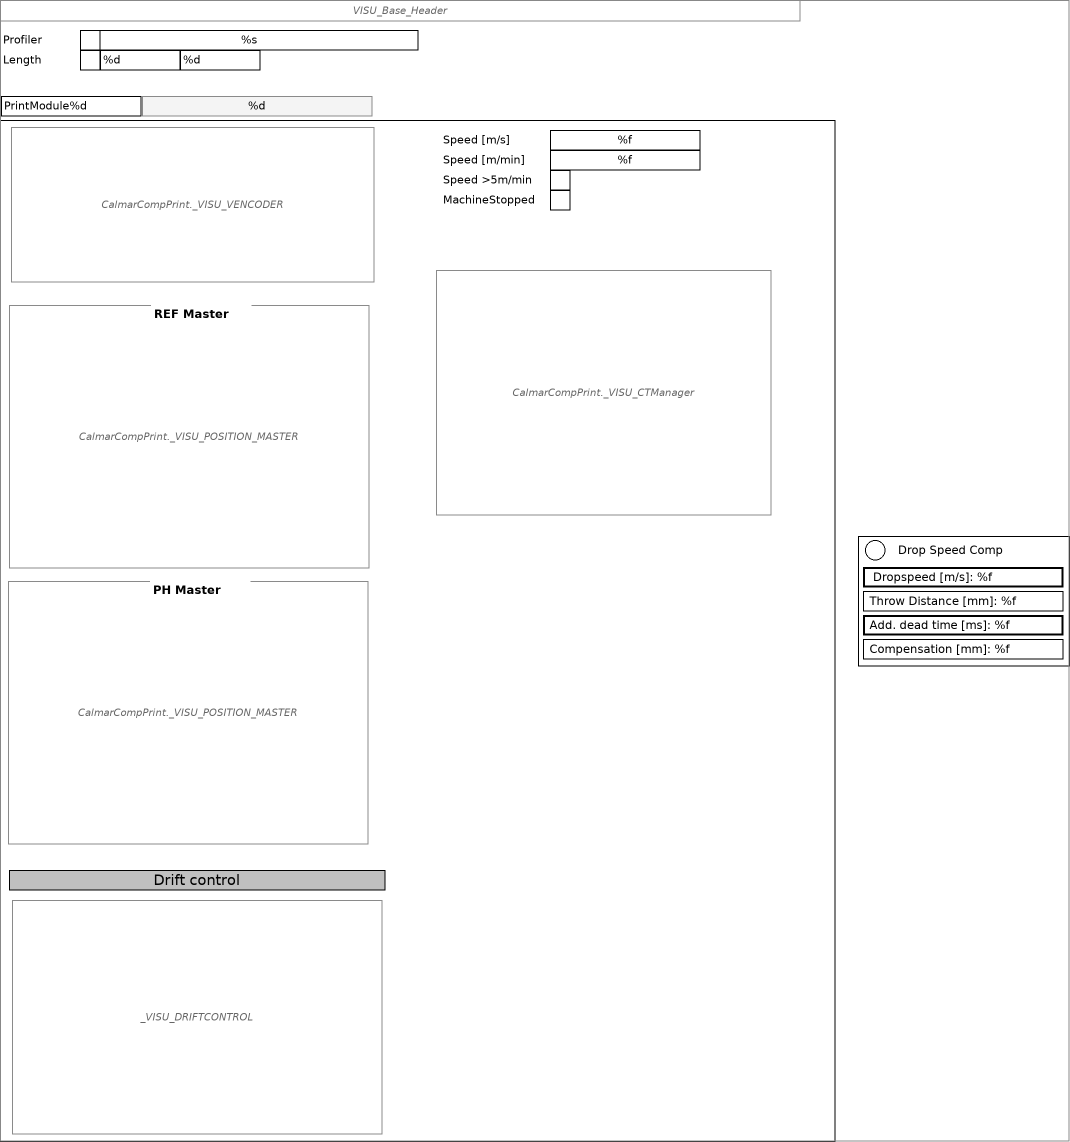
VISUALIZATION VISU_PrintDetails  // 1070x1142
    Rectangle (0,120 835x1022)
    Frame (9,305 360x263)
        shows CalmarCompPrint._VISU_POSITION_MASTER(m_Inst_Fb := PRG_PRINT.Fb_Ref_Master[PRG_PRINT.nSelectPmView])
    Frame (436,270 335x245)
        shows CalmarCompPrint._VISU_CTManager(m_Inst := PRG_PRINT.fBCTManager[PRG_PRINT.nSelectPmView])
    Rectangle (80,30 338x20), "%s", text variable: PRG_PRINT.fbProfiler.aProfilerData
    Rectangle (80,30 20x20)
        tap PRG_PRINT.fbProfiler.bReset
    Rectangle (151,304 100x20), "REF Master"
    Frame (8,581 360x263)
        shows CalmarCompPrint._VISU_POSITION_MASTER(m_Inst_Fb := PRG_PRINT.Fb_Ph_Master[PRG_PRINT.nSelectPmView])
    Rectangle (150,580 100x20), "PH Master"
    Scrollbar (142,96 230x20), "%d", text variable: PRG_PRINT.nSelectPmView
        p1057716461: PRG_PRINT.nSelectPmView
    Rectangle (1,96 140x20), "PrintModule%d", text variable: PRG_PRINT.nSelectPmView
    Frame (11,127 363x155)
        shows CalmarCompPrint._VISU_VENCODER(m_Inst := PRG_PRINT.fbVencoder[PRG_PRINT.nSelectPmView])
    Rectangle (550,130 150x20), "%f", text variable: PRG_PRINT.Fb_Ph_Master[PRG_PRINT.nSelectPmView].fO_Master_Speed
    Rectangle (440,130 110x20), "Speed [m/s]"
    Rectangle (550,150 150x20), "%f", text variable: PRG_PRINT.fL_SpeedInMpMin[PRG_PRINT.nSelectPmView]
    Rectangle (440,150 110x20), "Speed [m/min]"
    RoundedRectangle (550,170 20x20), colour toggle: PRG_PRINT.bL_MachineUpper5MpMin[PRG_PRINT.nSelectPmView]
    RoundedRectangle (550,190 20x20), colour toggle: PRG_PRINT.bL_MachineStopped[PRG_PRINT.nSelectPmView]
    Rectangle (440,170 110x20), "Speed >5m/min"
    Rectangle (440,190 110x20), "MachineStopped"
    Frame (12,900 370x234)
        shows _VISU_DRIFTCONTROL(mRef := PRG_PRINT.fB_DriftControl[PRG_PRINT.nSelectPmView])
    Rectangle (9,870 376x20), "Drift control"
    Frame (0,0 800x21)
        shows VISU_Base_Header()
    Rectangle (0,30 80x20), "Profiler"
    Rectangle (0,50 80x20), "Length"
    Rectangle (100,50 80x20), "%d", tooltip "Length in Machine", text variable: PRG_MACHINE.lL_SubstrateLenPx
    Rectangle (180,50 80x20), "%d", tooltip "Length in Job", text variable: PRG_MACHINE.lL_ImageDepthPx
    RoundedRectangle (80,50 20x20), tooltip "Length Missmatch", colour toggle: PRG_MACHINE.bL_MismatchLength
    Rectangle (858,536 212x130)
    Ellipse (865,540 20x20), colour toggle: PRG_PRINT.bL_UseSpeedCompensation
        toggle PRG_PRINT.bL_UseSpeedCompensation
    Rectangle (895,540 124x20), "Drop Speed Comp"
    Rectangle (863,567 200x20), "Dropspeed [m/s]: %f", text variable: PRG_PRINT.fL_DropSpeed
        OnMouseDown: write the text variable via Edit
    Rectangle (863,591 200x20), "Throw Distance [mm]: %f", text variable: PRG_PRINT.fL_PrintUnitElevation[1]
    Rectangle (863,639 200x20), "Compensation [mm]: %f", text variable: 1000 * PRG_PRINT.fL_SpeedComp[ePr_PU_UNIT_1]
    Rectangle (863,615 200x20), "Add. dead time [ms]: %f", text variable: PRG_PRINT.fL_DropSpeedAddTime
        OnMouseDown: write the text variable via Edit
END_VISUALIZATION

(* stored: Version 1.1.0.1, ProductVersion 3.1.4024.9
   Visu VISU_PrintDetails: Id {cefb1ae0-691a-4fb5-812f-b682a2a54c9e} *)
